(* Logix 5000 project; controller AI_2711_Studio5000 vendor 1 type 14 code 149 rev 32.11; software revision 32.03 *)

TASK MainTask (continuous, watchdog 500 ms) : Balancas

MODULES
   Local : vendor 1 type 14 code 149 (Compact 0, rev 32.11)
      Discrete_IO : Embedded (Compact 1, rev 3.1, Output RPI 20 ms)
      BL04 : vendor 90 type 0 code 46 (Ethernet 192.168.1.53, rev 1.5, StandardDataDriven RPI 10 ms)
           BL04:I.Data[3]   // Tara
           BL04:I.Data[2]   // Peso Bruto ou Liquido
           BL04:I.Data[1].0   // Casas Decimais
           BL04:I.Data[1].1   // Casas Decimais
           BL04:I.Data[1].2   // Casas Decimais
           BL04:I.Data[1].4   // 1 = Variação do peso igual ou acima do valor configurado em MOV
           BL04:I.Data[1]   // Bits de Status
           BL04:I.Data[1].13   // 1 = Vazia
           BL04:I.Data[1].7   // 0 = Peso Bruto / 1 = Peso Liquido
           BL04:I.Data[1].9   // Unidade
           BL04:I.Data[1].10   // Unidade
           BL04:I.Data[1].12   // 1 = Tara Negativa
           BL04:I.Data[1].8   // 1 = Erro
           BL04:I.Data[1].6   // 1 = Sobrecarga
           BL04:I.Data[1].5   // 1 = Saturação
           BL04:I.Data[1].3   // 1 = PesoNegativo
           BL04:I.Data[1].14   // 1 = Calibração
           BL04:I.Data[1].11   // 1 = Variação do peso igual ou acima do valor configurado em PMOV
END_MODULES

VAR_GLOBAL   (* controller tags *)
   BL04_PesoBruto : REAL;
   BL04_PesoOK : BOOL := 1;
END_VAR

PROGRAM Balancas   (* main routine Principal *)

ROUTINE BL04   (* ladder *)
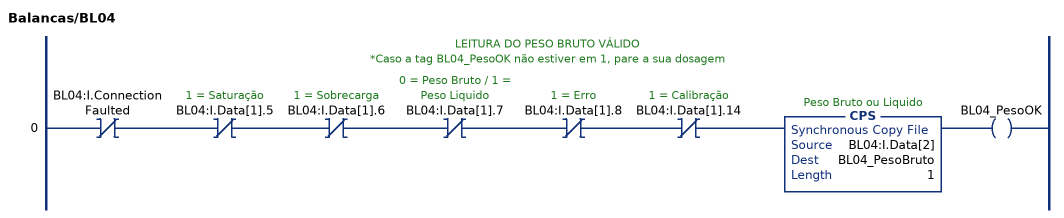
   // LEITURA DO PESO BRUTO VÁLIDO
   // *Caso a tag BL04_PesoOK não estiver em 1, pare a sua dosagem
   0: XIO(BL04:I.ConnectionFaulted)XIO(BL04:I.Data[1].5)XIO(BL04:I.Data[1].6)XIO(BL04:I.Data[1].7)XIO(BL04:I.Data[1].8)XIO(BL04:I.Data[1].14)CPS(BL04:I.Data[2],BL04_PesoBruto,1)OTE(BL04_PesoOK);
END_ROUTINE

ROUTINE Principal   (* ladder *)
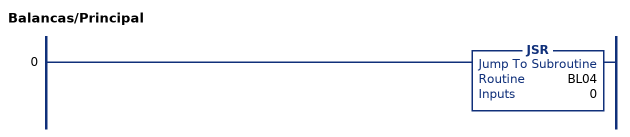
   0: JSR(BL04,0);
END_ROUTINE
END_PROGRAM
